{attribute addProperty BoxType "EL6002-0000-0019"}
{attribute addProperty Id "StatusAT %I*Status_A3013EBE8Data_InAT %I*ARRAY[0..21] OF USINT22"}
{attribute addProperty CRC "3350509587"}
{attribute addProperty SizeInBites "240"}
{attribute addProperty SizeInBytes "30"}
TYPE COM_TxPDO_Map_Inputs_Channel_F2FBC98A :
STRUCT
	{attribute addProperty Name "Status"}
	Status AT %I* : Status_A3013EBE;
	{attribute addProperty Name "Data_In"}
	Data_In AT %I* : ARRAY[0..21] OF USINT;
END_STRUCT
END_TYPE

(* stored: Version 1.2.0.0, ProductVersion 3.1.4024.9
   DUT COM_TxPDO_Map_Inputs_Channel_F2FBC98A: Id {de847c08-4e82-41fe-9342-049149deceb7} *)
